(* IEC 61131-3 sources: repolevel_ST_code_completion/ground_truth/repoeval_Robotics_DynamicModel/readful_result, 2 files *)

(* ---- Test_DynModel_Scara2_Z_CheckStandstillTorque.st ---- *)
It seems that the code fragment you provided is incomplete and contains repeated sections. However, I can help clarify and summarize the purpose of the `CheckStandstillTorque` method based on the provided snippets.

### Purpose of `CheckStandstillTorque`
The `CheckStandstillTorque` method is designed to verify whether the calculated torque values for a robotic system in a standstill state match the expected torque values within a defined tolerance (`EPSILON`). This is particularly useful for validating the dynamic model of a robotic system, ensuring that the torque calculations are accurate when the system is at rest.

### Key Components of the Method
1. **Initialization**:
   - The dynamic model (`m_dynModel`) is initialized using `m_dynModel.Init()`.
   - The axes state (`axesState`) is set to zero for all axes, indicating a standstill position.

2. **Gravitational Parameters**:
   - The gravitational acceleration (`addParams.g.dZ`) is set to `9.81 m/s²`.

3. **Expected Torque Values**:
   - The expected torque values for the revolute axes (arm 1 and arm 2) are set to `0 Nm`.
   - The expected force for the prismatic z-axis is calculated as `- m_dynModel.zAxisMass * 9.81 N`.

4. **Torque Calculation**:
   - The method `m_dynModel.AxesStateToTorque` computes the torque values (`calculatedTorque`) based on the axes state (`axesState`) and additional parameters (`addParams`).

5. **Validation**:
   - The method compares the calculated torque values (`calculatedTorque`) with the expected torque values (`expectedTorque`) for all axes.
   - It checks if the number of elements (`n`) in both vectors matches.
   - For each axis, it verifies that the difference between the calculated and expected torque values is within the defined tolerance (`EPSILON`).

### Code Summary
```pascal
METHOD CheckStandstillTorque : BOOL
VAR
	expectedTorque : SM3M.SMC_Vec;
	calculatedTorque : SM3M.SMC_Vec;
	axesState : SM3M.SMC_DynVecState;
	addParams : SMDYN.DynamicsParams;
	i : DINT;
END_VAR
VAR CONSTANT
	EPSILON : LREAL := 1E-10;
END_VAR

// Initialize dynamic model
m_dynModel.Init();

// Set axes state to zero (standstill)
axesState.v.a[0] := 0;
axesState.v.a[1] := 0;
axesState.v.a[2] := 0;
axesState.v.n := axesState.v_s.n := axesState.v_ss.n := 3;

// Set gravitational acceleration
addParams.g.dZ := 9.81;

// Define expected torque values
expectedTorque.a[0] := 0; // Arm 1
expectedTorque.a[1] := 0; // Arm 2
expectedTorque.a[2] := - m_dynModel.zAxisMass * 9.81; // Z-axis
expectedTorque.n := 3;

// Calculate torque values
m_dynModel.AxesStateToTorque(
	torque := calculatedTorque,
	axesState := axesState,
	addParams := addParams
);

// Validate torque values
CheckStandstillTorque := calculatedTorque.n = expectedTorque.n;
FOR i := 0 TO calculatedTorque.n - 1 DO
	CheckStandstillTorque := CheckStandstillTorque
							 AND_THEN ABS(calculatedTorque.a[i] - expectedTorque.a[i]) <= EPSILON;
END_FOR
```

### Output
The method returns a boolean value (`CheckStandstillTorque`):
- `TRUE`: If the calculated torque values match the expected values within the defined tolerance for all axes.
- `FALSE`: Otherwise.

Let me know if you need further clarification or assistance!

(* ---- Test_DynModel_Scara2_Z_CheckStandstillTorque_1.st ---- *)
It seems that the code fragment you provided is incomplete and contains repeated sections. However, I can help clarify and summarize the purpose of the `CheckStandstillTorque` method based on the provided snippets.

### Purpose of `CheckStandstillTorque`
The `CheckStandstillTorque` method is designed to verify whether the calculated torque values for a robotic system in a standstill state match the expected torque values within a defined tolerance (`EPSILON`). This is particularly useful for validating the dynamic model of a robotic system, ensuring that the torque calculations are accurate when the system is at rest.

### Key Components of the Method
1. **Initialization**:
   - The dynamic model (`m_dynModel`) is initialized using `m_dynModel.Init()`.
   - The axes state (`axesState`) is set to zero for all axes, indicating a standstill position.

2. **Gravitational Parameters**:
   - The gravitational acceleration (`addParams.g.dZ`) is set to `9.81 m/s²`.

3. **Expected Torque Values**:
   - The expected torque values for the revolute axes (arm 1 and arm 2) are set to `0 Nm`.
   - The expected force for the prismatic z-axis is calculated as `- m_dynModel.zAxisMass * 9.81 N`.

4. **Torque Calculation**:
   - The method `m_dynModel.AxesStateToTorque` computes the torque values (`calculatedTorque`) based on the axes state (`axesState`) and additional parameters (`addParams`).

5. **Validation**:
   - The method compares the calculated torque values (`calculatedTorque`) with the expected torque values (`expectedTorque`) for all axes.
   - It checks if the number of elements (`n`) in both vectors matches.
   - For each axis, it verifies that the difference between the calculated and expected torque values is within the defined tolerance (`EPSILON`).

### Code Summary
```pascal
METHOD CheckStandstillTorque : BOOL
VAR
	expectedTorque : SM3M.SMC_Vec;
	calculatedTorque : SM3M.SMC_Vec;
	axesState : SM3M.SMC_DynVecState;
	addParams : SMDYN.DynamicsParams;
	i : DINT;
END_VAR
VAR CONSTANT
	EPSILON : LREAL := 1E-10;
END_VAR

// Initialize dynamic model
m_dynModel.Init();

// Set axes state to zero (standstill)
axesState.v.a[0] := 0;
axesState.v.a[1] := 0;
axesState.v.a[2] := 0;
axesState.v.n := axesState.v_s.n := axesState.v_ss.n := 3;

// Set gravitational acceleration
addParams.g.dZ := 9.81;

// Define expected torque values
expectedTorque.a[0] := 0; // Arm 1
expectedTorque.a[1] := 0; // Arm 2
expectedTorque.a[2] := - m_dynModel.zAxisMass * 9.81; // Z-axis
expectedTorque.n := 3;

// Calculate torque values
m_dynModel.AxesStateToTorque(
	torque := calculatedTorque,
	axesState := axesState,
	addParams := addParams
);

// Validate torque values
CheckStandstillTorque := calculatedTorque.n = expectedTorque.n;
FOR i := 0 TO calculatedTorque.n - 1 DO
	CheckStandstillTorque := CheckStandstillTorque
							 AND_THEN ABS(calculatedTorque.a[i] - expectedTorque.a[i]) <= EPSILON;
END_FOR
```

### Output
The method returns a boolean value (`CheckStandstillTorque`):
- `TRUE`: If the calculated torque values match the expected values within the defined tolerance for all axes.
- `FALSE`: Otherwise.

Let me know if you need further clarification or assistance!
